REGION Network 20: UNLOCK
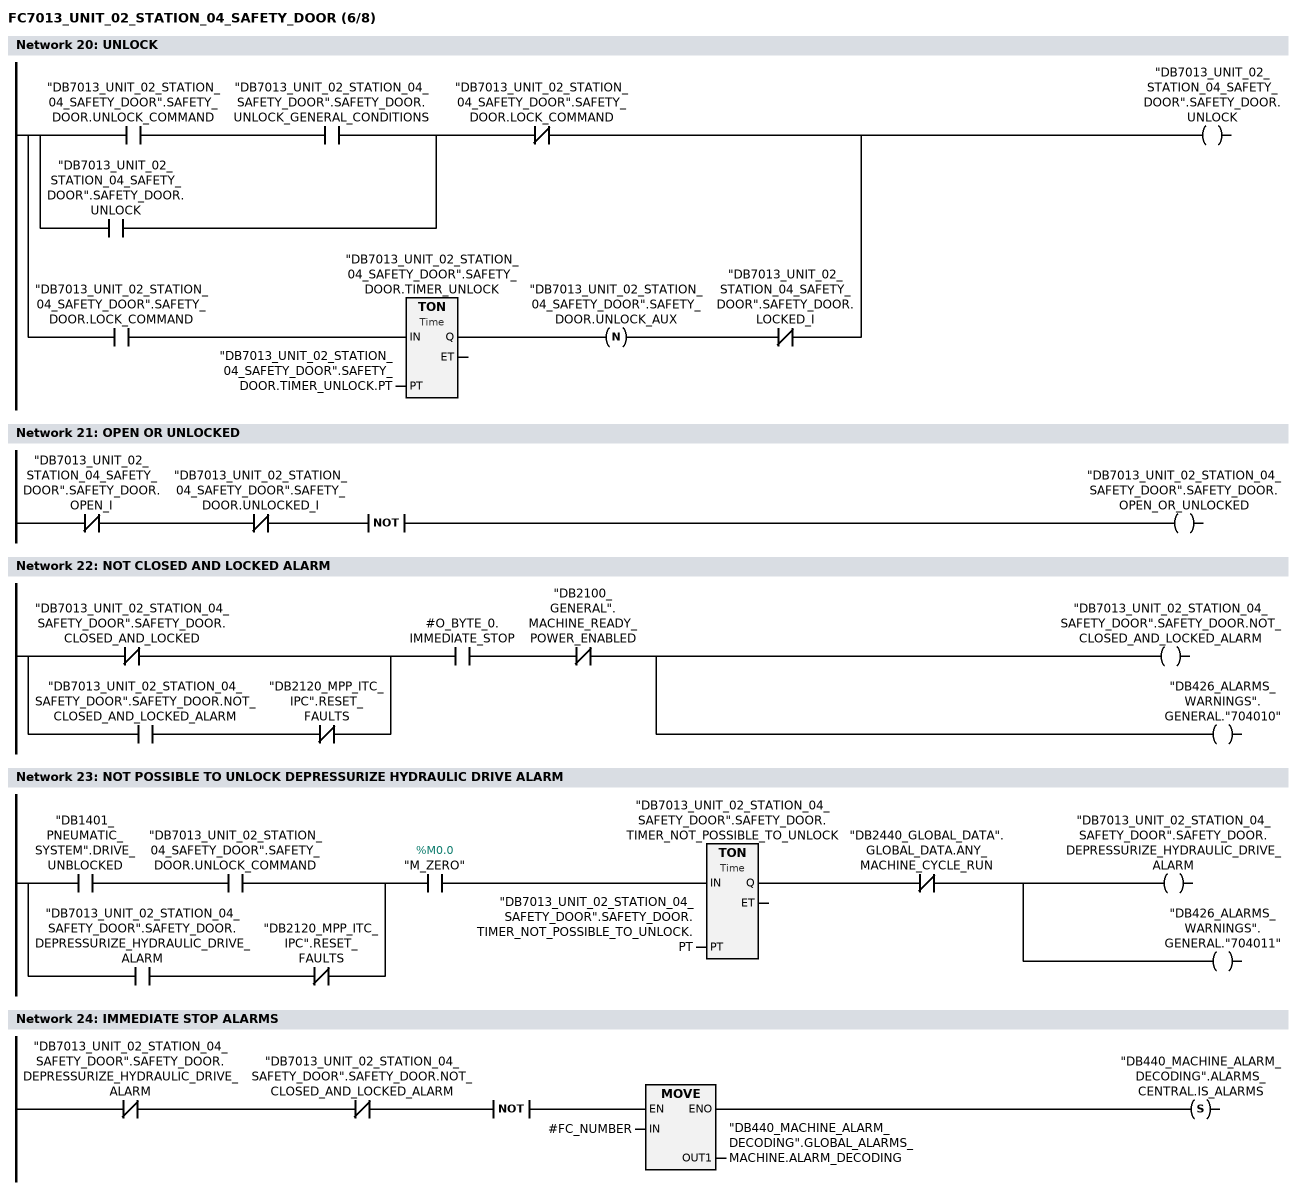
   RUNG wire#powerrail
      Contact( "DB7013_UNIT_02_STATION_04_SAFETY_DOOR".SAFETY_DOOR.UNLOCK_COMMAND )
      Contact( "DB7013_UNIT_02_STATION_04_SAFETY_DOOR".SAFETY_DOOR.UNLOCK_GENERAL_CONDITIONS )
      wire#w1
      I_Contact( "DB7013_UNIT_02_STATION_04_SAFETY_DOOR".SAFETY_DOOR.LOCK_COMMAND )
      wire#w2
      Coil( "DB7013_UNIT_02_STATION_04_SAFETY_DOOR".SAFETY_DOOR.UNLOCK )
   END_RUNG
   RUNG wire#powerrail
      Contact( "DB7013_UNIT_02_STATION_04_SAFETY_DOOR".SAFETY_DOOR.UNLOCK )
   END_RUNG wire#w1
   RUNG wire#powerrail
      Contact( "DB7013_UNIT_02_STATION_04_SAFETY_DOOR".SAFETY_DOOR.LOCK_COMMAND )
      { S7_Templates := "time_type := Time" } "DB7013_UNIT_02_STATION_04_SAFETY_DOOR".SAFETY_DOOR.TIMER_UNLOCK.TON(pt := "DB7013_UNIT_02_STATION_04_SAFETY_DOOR".SAFETY_DOOR.TIMER_UNLOCK.PT, et =>)
      N_Trig( "DB7013_UNIT_02_STATION_04_SAFETY_DOOR".SAFETY_DOOR.UNLOCK_AUX )
      I_Contact( "DB7013_UNIT_02_STATION_04_SAFETY_DOOR".SAFETY_DOOR.LOCKED_I )
   END_RUNG wire#w2
   // the same network as SCL:
   "DB7013_UNIT_02_STATION_04_SAFETY_DOOR".SAFETY_DOOR.TIMER_UNLOCK.TON(IN := "DB7013_UNIT_02_STATION_04_SAFETY_DOOR".SAFETY_DOOR.LOCK_COMMAND,
                           PT := "DB7013_UNIT_02_STATION_04_SAFETY_DOOR".SAFETY_DOOR.TIMER_UNLOCK.PT);
   #_w1 := NOT "DB7013_UNIT_02_STATION_04_SAFETY_DOOR".SAFETY_DOOR.TIMER_UNLOCK.Q AND "DB7013_UNIT_02_STATION_04_SAFETY_DOOR".SAFETY_DOOR.UNLOCK_AUX;   // falling edge
   "DB7013_UNIT_02_STATION_04_SAFETY_DOOR".SAFETY_DOOR.UNLOCK_AUX := "DB7013_UNIT_02_STATION_04_SAFETY_DOOR".SAFETY_DOOR.TIMER_UNLOCK.Q;
   "DB7013_UNIT_02_STATION_04_SAFETY_DOOR".SAFETY_DOOR.UNLOCK := ((("DB7013_UNIT_02_STATION_04_SAFETY_DOOR".SAFETY_DOOR.UNLOCK_COMMAND AND "DB7013_UNIT_02_STATION_04_SAFETY_DOOR".SAFETY_DOOR.UNLOCK_GENERAL_CONDITIONS) OR "DB7013_UNIT_02_STATION_04_SAFETY_DOOR".SAFETY_DOOR.UNLOCK) AND NOT "DB7013_UNIT_02_STATION_04_SAFETY_DOOR".SAFETY_DOOR.LOCK_COMMAND) OR (#_w1 AND NOT "DB7013_UNIT_02_STATION_04_SAFETY_DOOR".SAFETY_DOOR.LOCKED_I);
END_REGION

REGION Network 21: OPEN OR UNLOCKED
   RUNG wire#powerrail
      I_Contact( "DB7013_UNIT_02_STATION_04_SAFETY_DOOR".SAFETY_DOOR.OPEN_I )
      I_Contact( "DB7013_UNIT_02_STATION_04_SAFETY_DOOR".SAFETY_DOOR.UNLOCKED_I )
      Not()
      Coil( "DB7013_UNIT_02_STATION_04_SAFETY_DOOR".SAFETY_DOOR.OPEN_OR_UNLOCKED )
   END_RUNG
   // the same network as SCL:
   "DB7013_UNIT_02_STATION_04_SAFETY_DOOR".SAFETY_DOOR.OPEN_OR_UNLOCKED := NOT (NOT "DB7013_UNIT_02_STATION_04_SAFETY_DOOR".SAFETY_DOOR.OPEN_I AND NOT "DB7013_UNIT_02_STATION_04_SAFETY_DOOR".SAFETY_DOOR.UNLOCKED_I);
END_REGION

REGION Network 22: NOT CLOSED AND LOCKED ALARM
   RUNG wire#powerrail
      I_Contact( "DB7013_UNIT_02_STATION_04_SAFETY_DOOR".SAFETY_DOOR.CLOSED_AND_LOCKED )
      wire#w1
      Contact( #O_BYTE_0.IMMEDIATE_STOP )
      I_Contact( "DB2100_GENERAL".MACHINE_READY_POWER_ENABLED )
      wire#w2
      Coil( "DB7013_UNIT_02_STATION_04_SAFETY_DOOR".SAFETY_DOOR.NOT_CLOSED_AND_LOCKED_ALARM )
   END_RUNG
   RUNG wire#powerrail
      Contact( "DB7013_UNIT_02_STATION_04_SAFETY_DOOR".SAFETY_DOOR.NOT_CLOSED_AND_LOCKED_ALARM )
      I_Contact( "DB2120_MPP_ITC_IPC".RESET_FAULTS )
   END_RUNG wire#w1
   RUNG wire#w2
      Coil( "DB426_ALARMS_WARNINGS".GENERAL."704010" )
   END_RUNG
   // the same network as SCL:
   "DB7013_UNIT_02_STATION_04_SAFETY_DOOR".SAFETY_DOOR.NOT_CLOSED_AND_LOCKED_ALARM := (NOT "DB7013_UNIT_02_STATION_04_SAFETY_DOOR".SAFETY_DOOR.CLOSED_AND_LOCKED OR ("DB7013_UNIT_02_STATION_04_SAFETY_DOOR".SAFETY_DOOR.NOT_CLOSED_AND_LOCKED_ALARM AND NOT "DB2120_MPP_ITC_IPC".RESET_FAULTS)) AND #O_BYTE_0.IMMEDIATE_STOP AND NOT "DB2100_GENERAL".MACHINE_READY_POWER_ENABLED;
   "DB426_ALARMS_WARNINGS".GENERAL."704010" := "DB7013_UNIT_02_STATION_04_SAFETY_DOOR".SAFETY_DOOR.NOT_CLOSED_AND_LOCKED_ALARM;
END_REGION

REGION Network 23: NOT POSSIBLE TO UNLOCK DEPRESSURIZE HYDRAULIC DRIVE ALARM
   RUNG wire#powerrail
      Contact( "DB1401_PNEUMATIC_SYSTEM".DRIVE_UNBLOCKED )
      Contact( "DB7013_UNIT_02_STATION_04_SAFETY_DOOR".SAFETY_DOOR.UNLOCK_COMMAND )
      wire#w1
      Contact( "M_ZERO" )
      { S7_Templates := "time_type := Time" } "DB7013_UNIT_02_STATION_04_SAFETY_DOOR".SAFETY_DOOR.TIMER_NOT_POSSIBLE_TO_UNLOCK.TON(pt := "DB7013_UNIT_02_STATION_04_SAFETY_DOOR".SAFETY_DOOR.TIMER_NOT_POSSIBLE_TO_UNLOCK.PT, et =>)
      I_Contact( "DB2440_GLOBAL_DATA".GLOBAL_DATA.ANY_MACHINE_CYCLE_RUN )
      wire#w2
      Coil( "DB7013_UNIT_02_STATION_04_SAFETY_DOOR".SAFETY_DOOR.DEPRESSURIZE_HYDRAULIC_DRIVE_ALARM )
   END_RUNG
   RUNG wire#powerrail
      Contact( "DB7013_UNIT_02_STATION_04_SAFETY_DOOR".SAFETY_DOOR.DEPRESSURIZE_HYDRAULIC_DRIVE_ALARM )
      I_Contact( "DB2120_MPP_ITC_IPC".RESET_FAULTS )
   END_RUNG wire#w1
   RUNG wire#w2
      Coil( "DB426_ALARMS_WARNINGS".GENERAL."704011" )
   END_RUNG
   // the same network as SCL:
   "DB7013_UNIT_02_STATION_04_SAFETY_DOOR".SAFETY_DOOR.TIMER_NOT_POSSIBLE_TO_UNLOCK.TON(IN := (("DB1401_PNEUMATIC_SYSTEM".DRIVE_UNBLOCKED AND "DB7013_UNIT_02_STATION_04_SAFETY_DOOR".SAFETY_DOOR.UNLOCK_COMMAND) OR ("DB7013_UNIT_02_STATION_04_SAFETY_DOOR".SAFETY_DOOR.DEPRESSURIZE_HYDRAULIC_DRIVE_ALARM AND NOT "DB2120_MPP_ITC_IPC".RESET_FAULTS)) AND "M_ZERO",
                           PT := "DB7013_UNIT_02_STATION_04_SAFETY_DOOR".SAFETY_DOOR.TIMER_NOT_POSSIBLE_TO_UNLOCK.PT);
   "DB7013_UNIT_02_STATION_04_SAFETY_DOOR".SAFETY_DOOR.DEPRESSURIZE_HYDRAULIC_DRIVE_ALARM := "DB7013_UNIT_02_STATION_04_SAFETY_DOOR".SAFETY_DOOR.TIMER_NOT_POSSIBLE_TO_UNLOCK.Q AND NOT "DB2440_GLOBAL_DATA".GLOBAL_DATA.ANY_MACHINE_CYCLE_RUN;
   "DB426_ALARMS_WARNINGS".GENERAL."704011" := "DB7013_UNIT_02_STATION_04_SAFETY_DOOR".SAFETY_DOOR.DEPRESSURIZE_HYDRAULIC_DRIVE_ALARM;
END_REGION

REGION Network 24: IMMEDIATE STOP ALARMS
   RUNG wire#powerrail
      I_Contact( "DB7013_UNIT_02_STATION_04_SAFETY_DOOR".SAFETY_DOOR.DEPRESSURIZE_HYDRAULIC_DRIVE_ALARM )
      I_Contact( "DB7013_UNIT_02_STATION_04_SAFETY_DOOR".SAFETY_DOOR.NOT_CLOSED_AND_LOCKED_ALARM )
      Not()
      { S7_GenerateENO := "TRUE" } Move(in := #FC_NUMBER, out1 => "DB440_MACHINE_ALARM_DECODING".GLOBAL_ALARMS_MACHINE.ALARM_DECODING)
      S_Coil( "DB440_MACHINE_ALARM_DECODING".ALARMS_CENTRAL.IS_ALARMS )
   END_RUNG
   // the same network as SCL:
   // ENO of a box is taken as its EN; it also drops when the box reports an error
   IF NOT (NOT "DB7013_UNIT_02_STATION_04_SAFETY_DOOR".SAFETY_DOOR.DEPRESSURIZE_HYDRAULIC_DRIVE_ALARM AND NOT "DB7013_UNIT_02_STATION_04_SAFETY_DOOR".SAFETY_DOOR.NOT_CLOSED_AND_LOCKED_ALARM) THEN
       "DB440_MACHINE_ALARM_DECODING".GLOBAL_ALARMS_MACHINE.ALARM_DECODING := #FC_NUMBER;
       "DB440_MACHINE_ALARM_DECODING".ALARMS_CENTRAL.IS_ALARMS := TRUE;
   END_IF;
END_REGION

REGION Network 25: UNLOCK REQUEST WARNING
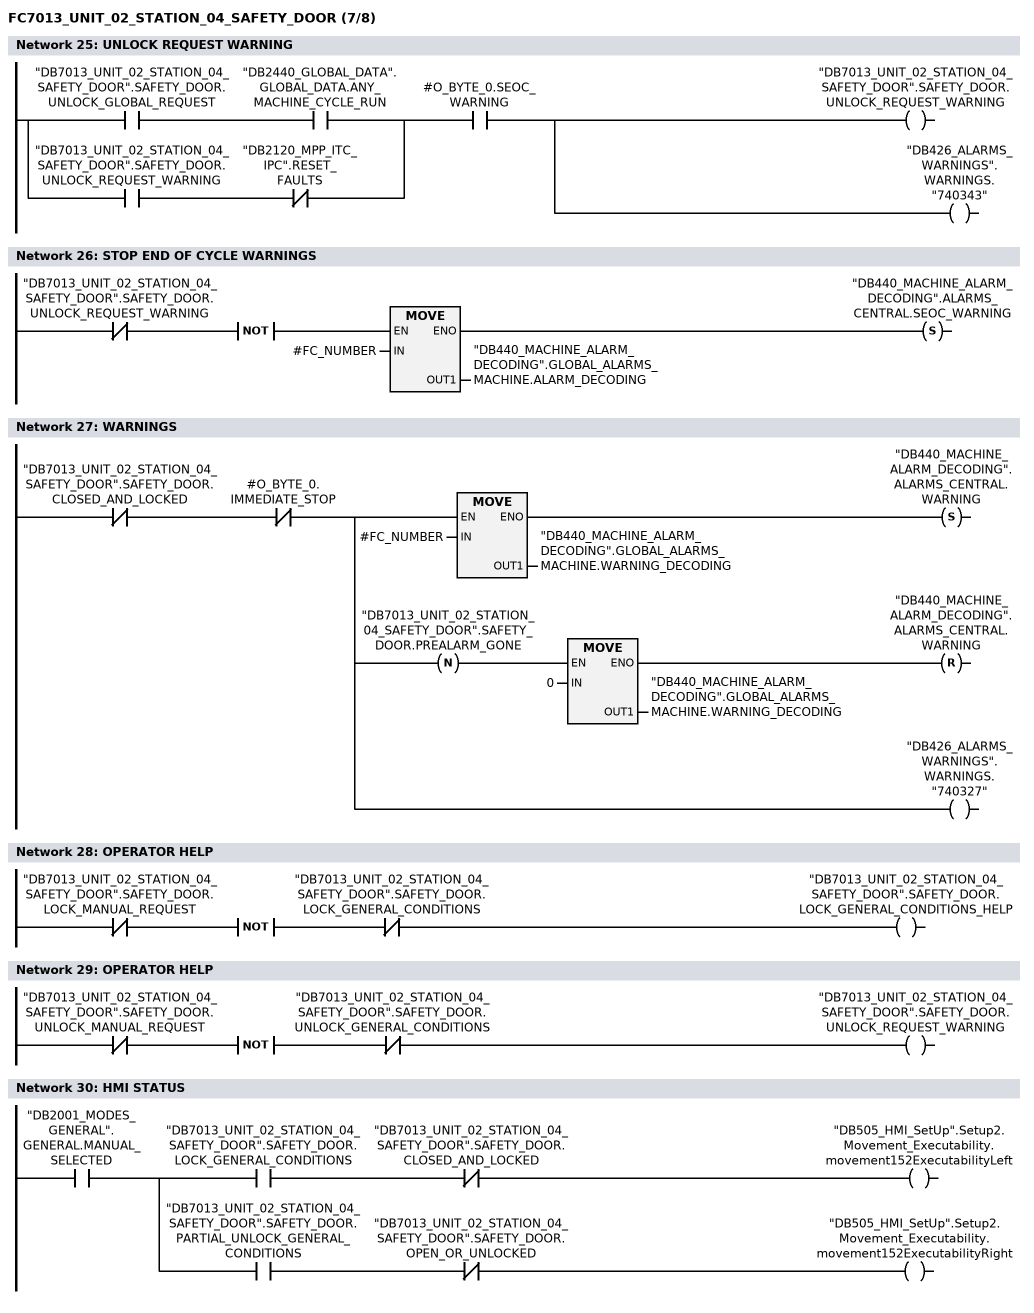
   RUNG wire#powerrail
      Contact( "DB7013_UNIT_02_STATION_04_SAFETY_DOOR".SAFETY_DOOR.UNLOCK_GLOBAL_REQUEST )
      Contact( "DB2440_GLOBAL_DATA".GLOBAL_DATA.ANY_MACHINE_CYCLE_RUN )
      wire#w1
      Contact( #O_BYTE_0.SEOC_WARNING )
      wire#w2
      Coil( "DB7013_UNIT_02_STATION_04_SAFETY_DOOR".SAFETY_DOOR.UNLOCK_REQUEST_WARNING )
   END_RUNG
   RUNG wire#powerrail
      Contact( "DB7013_UNIT_02_STATION_04_SAFETY_DOOR".SAFETY_DOOR.UNLOCK_REQUEST_WARNING )
      I_Contact( "DB2120_MPP_ITC_IPC".RESET_FAULTS )
   END_RUNG wire#w1
   RUNG wire#w2
      Coil( "DB426_ALARMS_WARNINGS".WARNINGS."740343" )
   END_RUNG
   // the same network as SCL:
   "DB7013_UNIT_02_STATION_04_SAFETY_DOOR".SAFETY_DOOR.UNLOCK_REQUEST_WARNING := (("DB7013_UNIT_02_STATION_04_SAFETY_DOOR".SAFETY_DOOR.UNLOCK_GLOBAL_REQUEST AND "DB2440_GLOBAL_DATA".GLOBAL_DATA.ANY_MACHINE_CYCLE_RUN) OR ("DB7013_UNIT_02_STATION_04_SAFETY_DOOR".SAFETY_DOOR.UNLOCK_REQUEST_WARNING AND NOT "DB2120_MPP_ITC_IPC".RESET_FAULTS)) AND #O_BYTE_0.SEOC_WARNING;
   "DB426_ALARMS_WARNINGS".WARNINGS."740343" := "DB7013_UNIT_02_STATION_04_SAFETY_DOOR".SAFETY_DOOR.UNLOCK_REQUEST_WARNING;
END_REGION

REGION Network 26: STOP END OF CYCLE WARNINGS
   RUNG wire#powerrail
      I_Contact( "DB7013_UNIT_02_STATION_04_SAFETY_DOOR".SAFETY_DOOR.UNLOCK_REQUEST_WARNING )
      Not()
      { S7_GenerateENO := "TRUE" } Move(in := #FC_NUMBER, out1 => "DB440_MACHINE_ALARM_DECODING".GLOBAL_ALARMS_MACHINE.ALARM_DECODING)
      S_Coil( "DB440_MACHINE_ALARM_DECODING".ALARMS_CENTRAL.SEOC_WARNING )
   END_RUNG
   // the same network as SCL:
   // ENO of a box is taken as its EN; it also drops when the box reports an error
   IF NOT (NOT "DB7013_UNIT_02_STATION_04_SAFETY_DOOR".SAFETY_DOOR.UNLOCK_REQUEST_WARNING) THEN
       "DB440_MACHINE_ALARM_DECODING".GLOBAL_ALARMS_MACHINE.ALARM_DECODING := #FC_NUMBER;
       "DB440_MACHINE_ALARM_DECODING".ALARMS_CENTRAL.SEOC_WARNING := TRUE;
   END_IF;
END_REGION

REGION Network 27: WARNINGS
   RUNG wire#powerrail
      I_Contact( "DB7013_UNIT_02_STATION_04_SAFETY_DOOR".SAFETY_DOOR.CLOSED_AND_LOCKED )
      I_Contact( #O_BYTE_0.IMMEDIATE_STOP )
      wire#w1
      { S7_GenerateENO := "TRUE" } Move(in := #FC_NUMBER, out1 => "DB440_MACHINE_ALARM_DECODING".GLOBAL_ALARMS_MACHINE.WARNING_DECODING)
      S_Coil( "DB440_MACHINE_ALARM_DECODING".ALARMS_CENTRAL.WARNING )
   END_RUNG
   RUNG wire#w1
      N_Trig( "DB7013_UNIT_02_STATION_04_SAFETY_DOOR".SAFETY_DOOR.PREALARM_GONE )
      { S7_GenerateENO := "TRUE" } Move(in := 0, out1 => "DB440_MACHINE_ALARM_DECODING".GLOBAL_ALARMS_MACHINE.WARNING_DECODING)
      R_Coil( "DB440_MACHINE_ALARM_DECODING".ALARMS_CENTRAL.WARNING )
   END_RUNG
   RUNG wire#w1
      Coil( "DB426_ALARMS_WARNINGS".WARNINGS."740327" )
   END_RUNG
   // the same network as SCL:
   // ENO of a box is taken as its EN; it also drops when the box reports an error
   #_w1 := NOT "DB7013_UNIT_02_STATION_04_SAFETY_DOOR".SAFETY_DOOR.CLOSED_AND_LOCKED AND NOT #O_BYTE_0.IMMEDIATE_STOP;
   IF #_w1 THEN
       "DB440_MACHINE_ALARM_DECODING".GLOBAL_ALARMS_MACHINE.WARNING_DECODING := #FC_NUMBER;
       "DB440_MACHINE_ALARM_DECODING".ALARMS_CENTRAL.WARNING := TRUE;
   END_IF;
   #_w2 := NOT #_w1 AND "DB7013_UNIT_02_STATION_04_SAFETY_DOOR".SAFETY_DOOR.PREALARM_GONE;   // falling edge
   "DB7013_UNIT_02_STATION_04_SAFETY_DOOR".SAFETY_DOOR.PREALARM_GONE := #_w1;
   IF #_w2 THEN
       "DB440_MACHINE_ALARM_DECODING".GLOBAL_ALARMS_MACHINE.WARNING_DECODING := 0;
       "DB440_MACHINE_ALARM_DECODING".ALARMS_CENTRAL.WARNING := FALSE;
   END_IF;
   "DB426_ALARMS_WARNINGS".WARNINGS."740327" := #_w1;
END_REGION

REGION Network 28: OPERATOR HELP
   RUNG wire#powerrail
      I_Contact( "DB7013_UNIT_02_STATION_04_SAFETY_DOOR".SAFETY_DOOR.LOCK_MANUAL_REQUEST )
      Not()
      I_Contact( "DB7013_UNIT_02_STATION_04_SAFETY_DOOR".SAFETY_DOOR.LOCK_GENERAL_CONDITIONS )
      Coil( "DB7013_UNIT_02_STATION_04_SAFETY_DOOR".SAFETY_DOOR.LOCK_GENERAL_CONDITIONS_HELP )
   END_RUNG
   // the same network as SCL:
   "DB7013_UNIT_02_STATION_04_SAFETY_DOOR".SAFETY_DOOR.LOCK_GENERAL_CONDITIONS_HELP := NOT (NOT "DB7013_UNIT_02_STATION_04_SAFETY_DOOR".SAFETY_DOOR.LOCK_MANUAL_REQUEST) AND NOT "DB7013_UNIT_02_STATION_04_SAFETY_DOOR".SAFETY_DOOR.LOCK_GENERAL_CONDITIONS;
END_REGION

REGION Network 29: OPERATOR HELP
   RUNG wire#powerrail
      I_Contact( "DB7013_UNIT_02_STATION_04_SAFETY_DOOR".SAFETY_DOOR.UNLOCK_MANUAL_REQUEST )
      Not()
      I_Contact( "DB7013_UNIT_02_STATION_04_SAFETY_DOOR".SAFETY_DOOR.UNLOCK_GENERAL_CONDITIONS )
      Coil( "DB7013_UNIT_02_STATION_04_SAFETY_DOOR".SAFETY_DOOR.UNLOCK_REQUEST_WARNING )
   END_RUNG
   // the same network as SCL:
   "DB7013_UNIT_02_STATION_04_SAFETY_DOOR".SAFETY_DOOR.UNLOCK_REQUEST_WARNING := NOT (NOT "DB7013_UNIT_02_STATION_04_SAFETY_DOOR".SAFETY_DOOR.UNLOCK_MANUAL_REQUEST) AND NOT "DB7013_UNIT_02_STATION_04_SAFETY_DOOR".SAFETY_DOOR.UNLOCK_GENERAL_CONDITIONS;
END_REGION

REGION Network 30: HMI STATUS
   RUNG wire#powerrail
      Contact( "DB2001_MODES_GENERAL".GENERAL.MANUAL_SELECTED )
      wire#w1
      Contact( "DB7013_UNIT_02_STATION_04_SAFETY_DOOR".SAFETY_DOOR.LOCK_GENERAL_CONDITIONS )
      I_Contact( "DB7013_UNIT_02_STATION_04_SAFETY_DOOR".SAFETY_DOOR.CLOSED_AND_LOCKED )
      Coil( "DB505_HMI_SetUp".Setup2.Movement_Executability.movement152ExecutabilityLeft )
   END_RUNG
   RUNG wire#w1
      Contact( "DB7013_UNIT_02_STATION_04_SAFETY_DOOR".SAFETY_DOOR.PARTIAL_UNLOCK_GENERAL_CONDITIONS )
      I_Contact( "DB7013_UNIT_02_STATION_04_SAFETY_DOOR".SAFETY_DOOR.OPEN_OR_UNLOCKED )
      Coil( "DB505_HMI_SetUp".Setup2.Movement_Executability.movement152ExecutabilityRight )
   END_RUNG
   // the same network as SCL:
   "DB505_HMI_SetUp".Setup2.Movement_Executability.movement152ExecutabilityLeft := "DB2001_MODES_GENERAL".GENERAL.MANUAL_SELECTED AND "DB7013_UNIT_02_STATION_04_SAFETY_DOOR".SAFETY_DOOR.LOCK_GENERAL_CONDITIONS AND NOT "DB7013_UNIT_02_STATION_04_SAFETY_DOOR".SAFETY_DOOR.CLOSED_AND_LOCKED;
   "DB505_HMI_SetUp".Setup2.Movement_Executability.movement152ExecutabilityRight := "DB2001_MODES_GENERAL".GENERAL.MANUAL_SELECTED AND "DB7013_UNIT_02_STATION_04_SAFETY_DOOR".SAFETY_DOOR.PARTIAL_UNLOCK_GENERAL_CONDITIONS AND NOT "DB7013_UNIT_02_STATION_04_SAFETY_DOOR".SAFETY_DOOR.OPEN_OR_UNLOCKED;
END_REGION

REGION Network 31: HMI STATUS
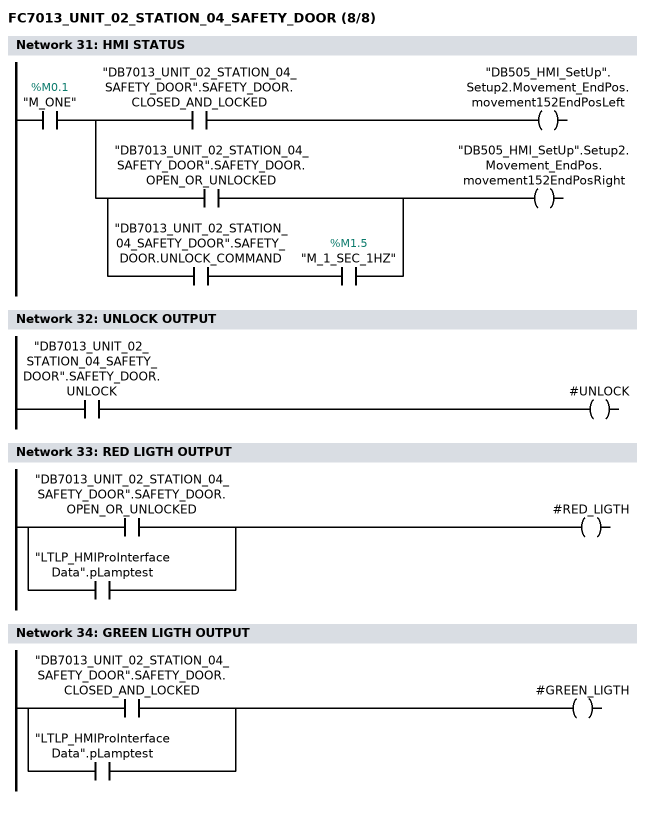
   RUNG wire#powerrail
      Contact( "M_ONE" )
      wire#w1
      Contact( "DB7013_UNIT_02_STATION_04_SAFETY_DOOR".SAFETY_DOOR.CLOSED_AND_LOCKED )
      Coil( "DB505_HMI_SetUp".Setup2.Movement_EndPos.movement152EndPosLeft )
   END_RUNG
   RUNG wire#w1
      Contact( "DB7013_UNIT_02_STATION_04_SAFETY_DOOR".SAFETY_DOOR.OPEN_OR_UNLOCKED )
      wire#w2
      Coil( "DB505_HMI_SetUp".Setup2.Movement_EndPos.movement152EndPosRight )
   END_RUNG
   RUNG wire#w1
      Contact( "DB7013_UNIT_02_STATION_04_SAFETY_DOOR".SAFETY_DOOR.UNLOCK_COMMAND )
      Contact( "M_1_SEC_1HZ" )
   END_RUNG wire#w2
   // the same network as SCL:
   "DB505_HMI_SetUp".Setup2.Movement_EndPos.movement152EndPosLeft := "M_ONE" AND "DB7013_UNIT_02_STATION_04_SAFETY_DOOR".SAFETY_DOOR.CLOSED_AND_LOCKED;
   "DB505_HMI_SetUp".Setup2.Movement_EndPos.movement152EndPosRight := "M_ONE" AND ("DB7013_UNIT_02_STATION_04_SAFETY_DOOR".SAFETY_DOOR.OPEN_OR_UNLOCKED OR ("DB7013_UNIT_02_STATION_04_SAFETY_DOOR".SAFETY_DOOR.UNLOCK_COMMAND AND "M_1_SEC_1HZ"));
END_REGION

REGION Network 32: UNLOCK OUTPUT
   RUNG wire#powerrail
      Contact( "DB7013_UNIT_02_STATION_04_SAFETY_DOOR".SAFETY_DOOR.UNLOCK )
      Coil( #UNLOCK )
   END_RUNG
   // the same network as SCL:
   #UNLOCK := "DB7013_UNIT_02_STATION_04_SAFETY_DOOR".SAFETY_DOOR.UNLOCK;
END_REGION

REGION Network 33: RED LIGTH OUTPUT
   RUNG wire#powerrail
      Contact( "DB7013_UNIT_02_STATION_04_SAFETY_DOOR".SAFETY_DOOR.OPEN_OR_UNLOCKED )
      wire#w1
      Coil( #RED_LIGTH )
   END_RUNG
   RUNG wire#powerrail
      Contact( "LTLP_HMIProInterfaceData".pLamptest )
   END_RUNG wire#w1
   // the same network as SCL:
   #RED_LIGTH := "DB7013_UNIT_02_STATION_04_SAFETY_DOOR".SAFETY_DOOR.OPEN_OR_UNLOCKED OR "LTLP_HMIProInterfaceData".pLamptest;
END_REGION

REGION Network 34: GREEN LIGTH OUTPUT
   RUNG wire#powerrail
      Contact( "DB7013_UNIT_02_STATION_04_SAFETY_DOOR".SAFETY_DOOR.CLOSED_AND_LOCKED )
      wire#w1
      Coil( #GREEN_LIGTH )
   END_RUNG
   RUNG wire#powerrail
      Contact( "LTLP_HMIProInterfaceData".pLamptest )
   END_RUNG wire#w1
   // the same network as SCL:
   #GREEN_LIGTH := "DB7013_UNIT_02_STATION_04_SAFETY_DOOR".SAFETY_DOOR.CLOSED_AND_LOCKED OR "LTLP_HMIProInterfaceData".pLamptest;
END_REGION
END_FUNCTION

FUNCTION "FC8007_UNIT_03_PART_STATUS_FULL_DEPTH" : Void   // FC8007, LAD
{ S7_Optimized_Access := 'TRUE' }
VERSION : 0.1
// stored: AutoNumber false, IsIECCheckEnabled false, SetENOAutomatically false, UDAEnableTagReadback false
BEGIN

REGION Network 1: FIXTURE 1 PART STATUS UNIT 01
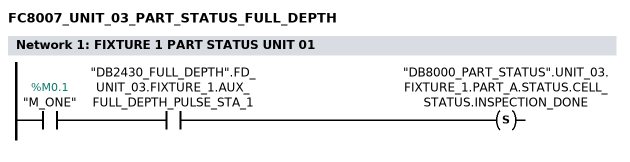
   RUNG wire#powerrail
      Contact( "M_ONE" )
      Contact( "DB2430_FULL_DEPTH".FD_UNIT_03.FIXTURE_1.AUX_FULL_DEPTH_PULSE_STA_1 )
      S_Coil( "DB8000_PART_STATUS".UNIT_03.FIXTURE_1.PART_A.STATUS.CELL_STATUS.INSPECTION_DONE )
   END_RUNG
   // the same network as SCL:
   IF "M_ONE" AND "DB2430_FULL_DEPTH".FD_UNIT_03.FIXTURE_1.AUX_FULL_DEPTH_PULSE_STA_1 THEN
       "DB8000_PART_STATUS".UNIT_03.FIXTURE_1.PART_A.STATUS.CELL_STATUS.INSPECTION_DONE := TRUE;
   END_IF;
END_REGION
END_FUNCTION

FUNCTION_BLOCK "FB2105_PSE200U_SITOP"
{ S7_Optimized_Access := 'FALSE' }
AUTHOR : DFCS
FAMILY : SITOP
NAME : PSE200U
VERSION : 2.3
   VAR_INPUT 
      impulse : Bool;
      reset : Bool;
   END_VAR

   VAR_OUTPUT 
      done : Bool;
      busy : Bool;
      channelState : Byte;
      status : Word;
      error : Bool;
   END_VAR

   VAR 
      statImpulseOld : Bool;
      statResetOld : Bool;
      statTimeSaver : Struct
         TimeTckRisingEdge : Time;
         TimeTckFallingEdge : Time;
         RisingEdgeDetected : Bool;
         FallingEdgeDetected : Bool;
         stateEdge : Int;
      END_STRUCT;
      statDeltaTimeImpulse : Time;
      statDeltaTimePause : Time;
      statStartImpulseDetected : Bool;
      statImpulseDetected : Bool;
      statChannelState : Byte;
      statChannelStateBool { ExternalAccessible := 'False'; ExternalVisible := 'False'; ExternalWritable := 'False'} AT statChannelState : Array[0..7] of Bool;
      statTimePauseSave0 : Time;
      statTimePauseSave1 : Time;
      statTimePauseSave2 : Time;
      statTimePauseSave3 : Time;
      statTimePauseSave4 : Time;
      statTimeImpulseSave0 : Time;
      statTimeImpulseSave1 : Time;
      statTimeImpulseSave2 : Time;
      statTimeImpulseSave3 : Time;
      statTimeImpulseSave4 : Time;
      statFrameImulseDetected : Bool;
      statNumberOfImpulses : Int;
      statChannelActive1 : Bool;
      statChannelActive2 : Bool;
      statChannelActive3 : Bool;
      statChannelActive4 : Bool;
      statCountChannelPos : Int;
      statCurrentPos1 : Int;
      statCurrentPos2 : Int;
      statCurrentPos3 : Int;
      statCurrentPos4 : Int;
      statTimeToImpulse : Time;
      statTimePause : Time;
      statTimeImpulse : Time;
      statTimeFrame : Time;
      statFrameOk : Bool;
      statCycleTimeNok : Bool;
      statSysTime : Time;
      statSysTimeOld : Time;
      statDeltaSysTime : Time;
      instSysTimer {InstructionName := 'TON_TIME'; LibVersion := '1.0'} : TON_TIME;
      statSysTimerStart : Bool;
      statStatus : Word;
      statIndex : Int;
      statSysTimerRun : Time;
      instWatchDogTimerR {InstructionName := 'TON_TIME'; LibVersion := '1.0'} : TON_TIME;
      statWatchDogTimerStartR : Bool;
      statWatchDogTimerRunR : Time;
      instWatchDogTimerF {InstructionName := 'TON_TIME'; LibVersion := '1.0'} : TON_TIME;
      statWatchDogTimerStartF : Bool;
      statWatchDogTimerRunF : Time;
      statResetRequest : Bool;
   END_VAR

   VAR_TEMP 
      tempLatchTime : Time;
   END_VAR

   VAR CONSTANT 
      STATE_IDLE : Int := 0;
      STATE_EVALUATION : Int := 1;
      STATE_ERROR : Int := 2;
      TIME_FRAME_MAX : Time := T#2S_850MS;
      TIME_FRAME_MIN : Time := T#2S_650MS;
      TIME_STARTIMPULSE_MIN : Time := T#400MS;
      TIME_STARTIMPULSE_MAX : Time := T#600MS;
      TIME_IMPULSE_MIN : Time := T#150MS;
      TIME_IMPULSE_MAX : Time := T#350MS;
      TIME_PAUSE1_MIN : Time := T#150MS;
      TIME_PAUSE1_MAX : Time := T#350MS;
      TIME_PAUSE2_MIN : Time := T#650MS;
      TIME_PAUSE2_MAX : Time := T#850MS;
      TIME_PAUSE3_MIN : Time := T#1S_150MS;
      TIME_PAUSE3_MAX : Time := T#1S_350MS;
      TIME_PAUSE4_MIN : Time := T#1S_650MS;
      TIME_PAUSE4_MAX : Time := T#1S_850MS;
      TIME_PAUSE_FRAME_MIN : Time := T#2S_150MS;
      TIME_PAUSE_FRAME_MAX : Time := T#2S_350MS;
   END_VAR


BEGIN
	   
	    // Calculate cycle time
	    #statSysTime := TIME_TCK();
	    #statDeltaSysTime := #statSysTime - #statSysTimeOld;
	    
	    IF (#statDeltaSysTime < t#0ms)
	    THEN
	        #statDeltaSysTime := #statDeltaSysTime + T#2147483647ms;
	        
	        IF #statDeltaSysTime < t#0ms
	        THEN
	            #statCycleTimeNok := true;
	            #statSysTimeOld := #statSysTime;
	            RETURN;
	        ELSE
	            #statCycleTimeNok := false;
	        END_IF;
	        
	    ELSIF #statDeltaSysTime >= t#102ms
	    THEN
	        #statCycleTimeNok := true;
	        #statSysTimerStart := true;
	    ELSE
	        #statCycleTimeNok := false;
	        #statSysTimerStart := false;
	    END_IF;
	    
	    //REGION edgeDetection
	        
	        IF ((#reset = true)
	            AND (#statResetOld = false))
	        THEN
	            #statSysTimerStart := false;
	            #statWatchDogTimerStartR := false;
	            #statWatchDogTimerStartF := false;
	            #statResetRequest := true;
	            #statIndex := #STATE_IDLE;
	        END_IF;
	        
	        //Rising edge at impulse input
	        IF ((#impulse = True)
	            AND (#statImpulseOld = False))
	        THEN
	            #tempLatchTime := TIME_TCK();
	            #statTimeSaver.RisingEdgeDetected := true;
	            #statTimeSaver.stateEdge := 15;
	            #statTimeSaver.TimeTckRisingEdge := #tempLatchTime;
	            #statWatchDogTimerStartR := true;
	            #statWatchDogTimerStartF := false;
	            
	            IF (#busy = false) THEN
	        
	                #busy := true;
	                #done := false;
	                #error := false;
	                #status := 16#0000;
	            END_IF;
	
	            
	            IF #statCycleTimeNok = false
	                AND #statResetRequest = false
	            THEN
	                #statIndex := #STATE_EVALUATION;
	            END_IF;
	        END_IF;
	        
	        //Falling edge at impulse input
	        IF ((#impulse = False)
	            AND (#statImpulseOld = True))
	        THEN
	            #tempLatchTime := TIME_TCK();
	            #statTimeSaver.FallingEdgeDetected := true;
	            #statTimeSaver.stateEdge := 16;
	            #statTimeSaver.TimeTckFallingEdge := #tempLatchTime;
	            #statWatchDogTimerStartF:=true;
	            #statWatchDogTimerStartR:=false;
	            
	            IF #statCycleTimeNok = FALSE
	                AND #statResetRequest = false
	            THEN
	                #statIndex := #STATE_EVALUATION;
	            END_IF;
	        END_IF;
	        
	        
	    //END_REGION
	    
	    IF #statTimeSaver.FallingEdgeDetected = false AND
	        #statTimeSaver.RisingEdgeDetected = FALSE
	    THEN
	        #statWatchDogTimerStartR := true;
	        #statWatchDogTimerStartF := true;
	    END_IF;
	    
	    CASE #statIndex OF
	        #STATE_IDLE:  // IDLE_STATE
	            #done := false;
	            #error := false;
	            #busy := false;
	            #status := 16#0000;
	            #statStatus := 16#0000;
	            #channelState := 16#00;
	            #statChannelState := 16#00;
	            #statFrameOk := false;
	            #statCycleTimeNok := false;
	            #statStartImpulseDetected := false;
	            #statFrameImulseDetected := false;
	            #statResetRequest := false;
	            #statTimeSaver.RisingEdgeDetected:=false;
	            #statTimeSaver.FallingEdgeDetected:=false;
	            
	        #STATE_EVALUATION:  //State: impulse detection
	            
	            //Delta time calculation
	            IF ((#statTimeSaver.RisingEdgeDetected = True)
	                AND (#statTimeSaver.FallingEdgeDetected = True))
	            THEN
	                
	                IF #statTimeSaver.stateEdge = 15 //pos. edge, evaluate delta pause
	                THEN
	                    #statDeltaTimePause := #statTimeSaver.TimeTckRisingEdge - #statTimeSaver.TimeTckFallingEdge;
	                    
	                    IF (#statDeltaTimePause < t#0ms)
	                    THEN
	                        #statDeltaTimePause := #statDeltaTimePause + T#2147483647ms;
	                        
	                        IF (#statDeltaTimePause < t#0ms)
	                        THEN
	                            #statIndex := #STATE_IDLE;
	                            #statTimeSaver.FallingEdgeDetected := false;
	                            RETURN;
	                        END_IF;
	                        
	                    ELSIF (#statDeltaTimePause > #TIME_FRAME_MAX)
	                    THEN
	                        #statIndex := #STATE_IDLE;
	                        #statTimeSaver.FallingEdgeDetected := false;
	                        RETURN;
	                    END_IF;
	                    #statTimeSaver.FallingEdgeDetected := false;
	                END_IF;
	                
	                IF #statTimeSaver.stateEdge = 16 // neg. edge, evaluate delta impulse
	                THEN
	                    #statImpulseDetected := true;
	                    #statDeltaTimeImpulse := #statTimeSaver.TimeTckFallingEdge - #statTimeSaver.TimeTckRisingEdge;
	                    
	                    IF (#statDeltaTimeImpulse < t#0ms)
	                    THEN
	                        #statDeltaTimeImpulse := #statDeltaTimeImpulse + T#2147483647ms;
	                        
	                        IF (#statDeltaTimeImpulse < t#0ms)
	                        THEN
	                            #statIndex := #STATE_IDLE;
	                            #statTimeSaver.RisingEdgeDetected := false;
	                            RETURN;
	                        END_IF;
	                        
	                    ELSIF (#statDeltaTimeImpulse > #TIME_FRAME_MAX)
	                    THEN
	                        #statIndex := #STATE_IDLE;
	                        #statTimeSaver.RisingEdgeDetected := false;
	                        RETURN;
	                    END_IF;
	                    #statTimeSaver.RisingEdgeDetected := false;
	                END_IF;
	            END_IF;
	            
	            //Start bit detection
	            IF ((#statDeltaTimeImpulse >= #TIME_STARTIMPULSE_MIN)
	                AND (#statDeltaTimeImpulse <= #TIME_STARTIMPULSE_MAX))
	                AND (#statImpulseDetected = True)
	            THEN
	                #statImpulseDetected := False;
	                #statNumberOfImpulses := 0;
	                #statCountChannelPos := 0;
	                
	                IF #statCurrentPos1 = 0
	                THEN
	                    #statTimeImpulseSave1 := t#0ms;
	                    #statTimePauseSave1 := t#0ms;
	                END_IF;
	                
	                IF #statCurrentPos2 = 0
	                THEN
	                    #statTimeImpulseSave2 := t#0ms;
	                    #statTimePauseSave2 := t#0ms;
	                END_IF;
	                
	                IF #statCurrentPos3 = 0
	                THEN
	                    #statTimeImpulseSave3 := t#0ms;
	                    #statTimePauseSave3 := t#0ms;
	                END_IF;
	                
	                IF #statCurrentPos4 = 0
	                THEN
	                    #statTimeImpulseSave4 := t#0ms;
	                    #statTimePauseSave4 := t#0ms;
	                END_IF;
	                
	                #statTimePauseSave0 := #statDeltaTimePause;
	                #statTimeImpulseSave0 := #statDeltaTimeImpulse;
	                
	                // get time in sum of imulses
	                #statTimeImpulse := #statTimeImpulseSave0 + #statTimeImpulseSave1 + #statTimeImpulseSave2 + #statTimeImpulseSave3 + #statTimeImpulseSave4;
	                
	                //get time in sum of pauses
	                #statTimePause := #statTimePauseSave0 + #statTimePauseSave1 + #statTimePauseSave2 + #statTimePauseSave3 + #statTimePauseSave4;
	                
	                // get length of frame
	                #statTimeFrame := #statTimeImpulse + #statTimePause;
	                
	                IF (#statTimeFrame >= t#2650ms)
	                    AND (#statTimeFrame <= #TIME_FRAME_MAX)
	                    AND (#statTimeToImpulse <= #TIME_FRAME_MIN)
	                THEN
	                    #statFrameOk := true;
	                END_IF;
	                
	                IF #statFrameOk = TRUE
	                    AND #statCycleTimeNok = FALSE
	                THEN
	                    // Daten Ã¼bernehmen
	                    #done := true;
	                    #busy := false;
	                    #statFrameOk := false;
	                    
	                    IF #statChannelActive1 = true
	                    THEN
	                        #statChannelStateBool[0] := false;
	                    ELSE
	                        #statChannelStateBool[0] := true;
	                    END_IF;
	                    
	                    IF #statChannelActive2 = true
	                    THEN
	                        #statChannelStateBool[1] := false;
	                    ELSE
	                        #statChannelStateBool[1] := true;
	                    END_IF;
	                    
	                    IF #statChannelActive3 = true
	                    THEN
	                        #statChannelStateBool[2] := false;
	                    ELSE
	                        #statChannelStateBool[2] := true;
	                    END_IF;
	                    
	                    IF #statChannelActive4 = true
	                    THEN
	                        #statChannelStateBool[3] := false;
	                    ELSE
	                        #statChannelStateBool[3] := true;
	                    END_IF;
	                    
	                    #channelState := #statChannelState;
	                END_IF;
	                
	                
	                // channel 4 ok
	                IF (#statDeltaTimePause >= #TIME_PAUSE1_MIN) AND
	                    (#statDeltaTimePause <= #TIME_PAUSE1_MAX)
	                THEN
	                    #statChannelActive4 := true;
	                    // channel 4 ok not ok
	                ELSIF
	                    (#statDeltaTimePause >= #TIME_PAUSE2_MIN) AND
	                    (#statDeltaTimePause <= #TIME_PAUSE2_MAX)
	                THEN
	                    #statChannelActive4 := false;
	                    // channel 3 and 4 not ok    
	                ELSIF
	                    (#statDeltaTimePause >= #TIME_PAUSE3_MIN) AND
	                    (#statDeltaTimePause <= #TIME_PAUSE3_MAX)
	                THEN
	                    #statChannelActive3 := false;
	                    #statChannelActive4 := false;
	                    // channel 2, 3, 4 not ok
	                ELSIF
	                    (#statDeltaTimePause >= #TIME_PAUSE4_MIN) AND
	                    (#statDeltaTimePause <= #TIME_PAUSE4_MAX)
	                THEN
	                    #statChannelActive2 := false;
	                    #statChannelActive3 := false;
	                    #statChannelActive4 := false;
	                    // channel 1, 2, 3, 4 not ok
	                ELSIF
	                    (#statDeltaTimePause >= #TIME_PAUSE_FRAME_MIN) AND
	                    (#statDeltaTimePause <= #TIME_PAUSE_FRAME_MAX)
	                THEN
	                    #statChannelActive1 := false;
	                    #statChannelActive2 := false;
	                    #statChannelActive3 := false;
	                    #statChannelActive4 := false;
	                END_IF;
	                
	                #statCountChannelPos := 4;
	                
	                #statCurrentPos1 := 0;
	                #statCurrentPos2 := 0;
	                #statCurrentPos3 := 0;
	                #statCurrentPos4 := 0;
	                
	                // Imulse bit detection
	            ELSIF ((#statDeltaTimeImpulse >= #TIME_IMPULSE_MIN)
	                AND (#statDeltaTimeImpulse <= #TIME_IMPULSE_MAX))
	                AND (#statImpulseDetected = True)
	            THEN
	                #statImpulseDetected := False;
	                #statFrameImulseDetected := true;
	            END_IF;
	            
	            //Channel detection
	            
	            IF #statFrameImulseDetected = TRUE
	            THEN
	                #statFrameImulseDetected := FALSE;
	                
	                IF #statCountChannelPos = 4
	                THEN
	                    #statCurrentPos1 := #statCountChannelPos;
	                    #statTimeImpulseSave1 := #statDeltaTimeImpulse;
	                    #statTimePauseSave1 := #statDeltaTimePause;
	                    #statTimeToImpulse := t#0ms;
	                    #statTimeToImpulse := #statTimeToImpulse + #statDeltaTimeImpulse + #statDeltaTimePause;
	                    
	                    //channel 1 ok
	                    IF (#statDeltaTimePause >= #TIME_PAUSE1_MIN)
	                        AND (#statDeltaTimePause <= #TIME_PAUSE1_MAX)
	                    THEN
	                        #statChannelActive1 := true;
	                        #statCountChannelPos := 1; // Pos 1 detected
	                    END_IF;
	                    
	                    // channel 1 not ok
	                    IF (#statDeltaTimePause >= #TIME_PAUSE2_MIN)
	                        AND (#statDeltaTimePause <= #TIME_PAUSE2_MAX)
	                    THEN
	                        #statChannelActive1 := false;
	                        #statChannelActive2 := true;
	                        #statCountChannelPos := 2; // go to next Pos 2
	                    END_IF;
	                    
	                    // channel 1 and 2 not ok
	                    IF (#statDeltaTimePause >= #TIME_PAUSE3_MIN)
	                        AND (#statDeltaTimePause <= #TIME_PAUSE3_MAX)
	                    THEN
	                        #statChannelActive1 := false;
	                        #statChannelActive2 := false;
	                        #statChannelActive3 := true;
	                        #statCountChannelPos := 2; // go to next Pos 2
	                    END_IF;
	                    
	                    // channel 1, 2 and 3 not ok
	                    IF (#statDeltaTimePause >= #TIME_PAUSE4_MIN)
	                        AND (#statDeltaTimePause <= #TIME_PAUSE4_MAX)
	                    THEN
	                        #statChannelActive1 := false;
	                        #statChannelActive2 := false;
	                        #statChannelActive3 := FALSE;
	                        #statChannelActive4 := true;
	                        #statCountChannelPos := 0;
	                    END_IF;
	                ELSIF #statCountChannelPos = 1
	                THEN
	                    #statCurrentPos2 := #statCountChannelPos;
	                    #statTimeImpulseSave2 := #statDeltaTimeImpulse;
	                    #statTimePauseSave2 := #statDeltaTimePause;
	                    #statTimeToImpulse := #statTimeToImpulse + #statDeltaTimeImpulse + #statDeltaTimePause;
	                    
	                    IF (#statDeltaTimePause >= #TIME_PAUSE1_MIN)
	                        AND (#statDeltaTimePause <= #TIME_PAUSE1_MAX)
	                    THEN
	                        #statChannelActive2 := true;
	                        #statCountChannelPos := 2; // go to next pos 2
	                    END_IF;
	                    
	                    IF (#statDeltaTimePause >= #TIME_PAUSE2_MIN)
	                        AND (#statDeltaTimePause <= #TIME_PAUSE2_MAX)
	                    THEN
	                        #statChannelActive2 := false;
	                        #statChannelActive3 := true;
	                        #statCountChannelPos := 2; // go to next Pos 2
	                    END_IF;
	                    
	                    IF (#statDeltaTimePause >= #TIME_PAUSE3_MIN)
	                        AND (#statDeltaTimePause <= #TIME_PAUSE3_MAX)
	                    THEN
	                        #statChannelActive2 := false;
	                        #statChannelActive3 := false;
	                        #statChannelActive4 := true;
	                        #statCountChannelPos := 0;
	                    END_IF;
	                ELSIF #statCountChannelPos = 2
	                THEN
	                    #statCurrentPos3 := #statCountChannelPos;
	                    #statTimeImpulseSave3 := #statDeltaTimeImpulse;
	                    #statTimePauseSave3 := #statDeltaTimePause;
	                    #statTimeToImpulse := #statTimeToImpulse + #statDeltaTimeImpulse + #statDeltaTimePause;
	                    
	                    IF (#statDeltaTimePause >= #TIME_PAUSE1_MIN)
	                        AND (#statDeltaTimePause <= #TIME_PAUSE1_MAX)
	                    THEN
	                        #statChannelActive3 := true;
	                        #statCountChannelPos := 3; // go to next pos 3
	                    END_IF;
	                    
	                    IF (#statDeltaTimePause >= #TIME_PAUSE2_MIN)
	                        AND (#statDeltaTimePause <= #TIME_PAUSE2_MAX)
	                    THEN
	                        #statChannelActive3 := false;
	                        #statChannelActive4 := true;
	                        #statCountChannelPos := 0;
	                    END_IF;
	                ELSIF #statCountChannelPos = 3
	                THEN
	                    #statCurrentPos4 := #statCountChannelPos;
	                    #statTimeImpulseSave4 := #statDeltaTimeImpulse;
	                    #statTimePauseSave4 := #statDeltaTimePause;
	                    #statTimeToImpulse := #statTimeToImpulse + #statDeltaTimeImpulse + #statDeltaTimePause;
	                    
	                    IF (#statDeltaTimePause >= #TIME_PAUSE1_MIN)
	                        AND (#statDeltaTimePause <= #TIME_PAUSE1_MAX)
	                    THEN
	                        #statChannelActive4 := true;
	                    END_IF;
	                    #statCountChannelPos := 0; // go to pos 0
	                END_IF;
	            END_IF;
	            
	        #STATE_ERROR:
	            #error := true;
	            #busy := false;
	            #done := false;
	            #statSysTimerStart := false;
	            #statWatchDogTimerStartR := false;
	            #statWatchDogTimerStartF := false;
	            #status := #statStatus;
	            #statStatus := w#16#0000;
	            #statIndex := #STATE_IDLE;
	        ELSE  // Statement section ELSE
	            #statIndex := #STATE_IDLE;
	    END_CASE;
	    
	    #instWatchDogTimerR(IN := #statWatchDogTimerStartR,
	                       PT := t#6s);
	    #statWatchDogTimerRunR:= #instWatchDogTimerR.ET;
	    
	    
	    #instWatchDogTimerF(IN := #statWatchDogTimerStartF,
	                       PT := t#6s); 
	    #statWatchDogTimerRunF:= #instWatchDogTimerF.ET;
	          
	    #instSysTimer(IN := #statSysTimerStart,
	                  PT := T#4s);
	    #statSysTimerRun:= #instSysTimer.ET; 
	    
	    IF  (#instWatchDogTimerR.Q = true)
	        OR (#instWatchDogTimerF.Q = true)
	        THEN
	        #statIndex := #STATE_ERROR;
	        #statStatus := 16#8002;
	    END_IF;
	      
	    
	    IF #instSysTimer.Q=true
	    THEN
	        #statIndex := #STATE_ERROR;
	        #statStatus := 16#8001;
	    END_IF;
	    
	    //Edge control
	    #statImpulseOld := #impulse;
	    #statResetOld := #reset;
	    
	    // Cycle time control
	    #statSysTimeOld := #statSysTime;
	
END_FUNCTION_BLOCK

FUNCTION "FC450_ALARM_DECODING_WINCC" : Void
{ S7_Optimized_Access := 'TRUE' }
VERSION : 0.1
   VAR_TEMP 
      i : Int;
      val1 : Int;
   END_VAR


BEGIN
	// IF THE SIZE OF 'DB426_ALARMS_WARNINGS' IS CHANGED, THE MAXIMUM NUMBER OF WORDS 
	// IN THE 'FOR' LOOP AND THE NUMBER OF BYTES TRANSFERRED FROM 'DB426' TO 'DB429' WITH BLKMOV MUST BE UPDATED.
	
	#val1 := BLKMOV(SRCBLK := P#DB426.DBX0.0 BYTE 3874, DSTBLK => P#DB430.DBX0.0 BYTE 3874);
	
	FOR #i := 0 TO 1937 DO
	    "DB430_ALARMS_WARNINGS_WINCC_AUX".Alarms[#i] := SWAP("DB430_ALARMS_WARNINGS_WINCC_AUX".Alarms[#i]);
	END_FOR;
	
	#val1 := BLKMOV(SRCBLK := P#DB430.DBX0.0 Byte 3874, DSTBLK => P#DB429.DBX0.0 BYTE 3874);
END_FUNCTION

FUNCTION "FC2401_DTL_TO_UNIX_TIME_1" : Word
{ S7_Optimized_Access := 'TRUE' }
VERSION : 0.1
   VAR_INPUT 
      SYSTEM_TIME_DTL {InstructionName := 'DTL'; LibVersion := '1.0'} : DTL;
   END_VAR

   VAR_OUTPUT 
      UNIX_TIME_SEC : UDInt;
      UNIX_TIME_MSEC : UDInt;
   END_VAR

   VAR_TEMP 
      UNIX_TIME_UDINT : UDInt;
      NANOSEC_REAL : Real;
      MILISEC_REAL : Real;
   END_VAR

   VAR CONSTANT 
      DELTA_1970_1990 : UDInt := 631_152_000;
      SEC_PER_DAY : UDInt := 86400;
   END_VAR


BEGIN
	#FC2401_DTL_TO_UNIX_TIME_1 := 1;
	
	// Convert the system time value to Dint
	#UNIX_TIME_UDINT := (DATE_TO_UDINT(DTL_TO_DATE(#SYSTEM_TIME_DTL)) * #SEC_PER_DAY) + (TOD_TO_UDINT(DTL_TO_TOD(#SYSTEM_TIME_DTL)) / 1000) + #DELTA_1970_1990;
	
	// System nanoseconds converted to miliseconds
	#NANOSEC_REAL := UDINT_TO_REAL(#SYSTEM_TIME_DTL.NANOSECOND);
	#MILISEC_REAL := #NANOSEC_REAL / 1000000.0;
	
	// Conversion to  Output
	#UNIX_TIME_SEC := #UNIX_TIME_UDINT;
	#UNIX_TIME_MSEC := REAL_TO_UDINT(#MILISEC_REAL);
	
	// Done convertion
	#FC2401_DTL_TO_UNIX_TIME_1 := 0;
END_FUNCTION

FUNCTION_BLOCK "FB7238_VARIABLES_PLC_HMI_GENERAL"
{ S7_Optimized_Access := 'TRUE' }
VERSION : 0.1
   VAR_INPUT DB_SPECIFIC
      FEEDERS_MANUAL_MODE : Bool;
      FEEDERS_AUTO_MODE : Bool;
      HOPPERS_MANUAL_MODE : Bool;
      HOPPERS_AUTO_MODE : Bool;
   END_VAR

   VAR_OUTPUT 
      FEEDERS_MODE_STATE : Int;
      HOPPERS_MODE_STATE : Int;
   END_VAR


BEGIN
	(*
	PLC TO HMI
	*)
	// UNIT 01 MODE STATE
	IF #FEEDERS_MANUAL_MODE = TRUE  AND #FEEDERS_AUTO_MODE = FALSE THEN
	    // Statement section IF
	    #FEEDERS_MODE_STATE := 3;
	ELSIF #FEEDERS_MANUAL_MODE = FALSE  AND #FEEDERS_AUTO_MODE = TRUE THEN
	    #FEEDERS_MODE_STATE := 1;
	END_IF;
	
	
	// UNIT 02 MODE STATE
	IF #HOPPERS_MANUAL_MODE = TRUE AND #HOPPERS_AUTO_MODE = FALSE THEN
	    // Statement section IF
	    #HOPPERS_MODE_STATE := 3;
	ELSIF #HOPPERS_MANUAL_MODE = FALSE AND #HOPPERS_AUTO_MODE = TRUE THEN
	    #HOPPERS_MODE_STATE := 1;
	END_IF;
	
	
	
	
END_FUNCTION_BLOCK

DATA_BLOCK "DB21205_UNIT_01_COMBINER_MEDICOAT"   // DB21205
{ DB_Accessible_From_OPC_UA := 'FALSE' }
VERSION : 0.1
// stored: AutoNumber false, DBAccessibleFromOPCUA false, DBAccessibleFromWebserver true, InstanceOfName FB21200_POWDER_FLOW_SENSOR_MEDICOAT, InstanceOfType FB
"FB21200_POWDER_FLOW_SENSOR_MEDICOAT"
BEGIN
END_DATA_BLOCK

DATA_BLOCK "DB21206_UNIT_02_COMBINER_MEDICOAT"   // DB21206
{ DB_Accessible_From_OPC_UA := 'FALSE' }
VERSION : 0.1
// stored: AutoNumber false, DBAccessibleFromOPCUA false, DBAccessibleFromWebserver true, InstanceOfName FB21200_POWDER_FLOW_SENSOR_MEDICOAT, InstanceOfType FB
"FB21200_POWDER_FLOW_SENSOR_MEDICOAT"
BEGIN
END_DATA_BLOCK

DATA_BLOCK "DB21209_UNIT_01_LASER_HEAD_MEDICOAT"   // DB21209
{ DB_Accessible_From_OPC_UA := 'FALSE' }
VERSION : 0.1
// stored: AutoNumber false, DBAccessibleFromOPCUA false, DBAccessibleFromWebserver true, InstanceOfName FB21200_POWDER_FLOW_SENSOR_MEDICOAT, InstanceOfType FB
"FB21200_POWDER_FLOW_SENSOR_MEDICOAT"
BEGIN
END_DATA_BLOCK

DATA_BLOCK "DB21210_UNIT_02_LASER_HEAD_MEDICOAT"   // DB21210
{ DB_Accessible_From_OPC_UA := 'FALSE' }
VERSION : 0.1
// stored: AutoNumber false, DBAccessibleFromOPCUA false, DBAccessibleFromWebserver true, InstanceOfName FB21200_POWDER_FLOW_SENSOR_MEDICOAT, InstanceOfType FB
"FB21200_POWDER_FLOW_SENSOR_MEDICOAT"
BEGIN
END_DATA_BLOCK

DATA_BLOCK "DB21222_POWDER_FILLING_START_STOP_BY_CURRENT_DB"   // DB21222
{ DB_Accessible_From_OPC_UA := 'FALSE' }
VERSION : 0.1
// stored: AutoNumber false, DBAccessibleFromOPCUA false, DBAccessibleFromWebserver true, InstanceOfName FB21222_POWDER_FILLING_START_STOP_BY_CURRENT, InstanceOfType FB
"FB21222_POWDER_FILLING_START_STOP_BY_CURRENT"
BEGIN
END_DATA_BLOCK

DATA_BLOCK "DB21225_HOPPER_1_POWDER_FILLING_START_STOP_BY_CURRENT_DB"   // DB21225
{ DB_Accessible_From_OPC_UA := 'FALSE' }
VERSION : 0.1
// stored: AutoNumber false, DBAccessibleFromOPCUA false, DBAccessibleFromWebserver true, InstanceOfName FB21222_POWDER_FILLING_START_STOP_BY_CURRENT, InstanceOfType FB
"FB21222_POWDER_FILLING_START_STOP_BY_CURRENT"
BEGIN
END_DATA_BLOCK

DATA_BLOCK "DB21226_HOPPER_2_POWDER_FILLING_START_STOP_BY_CURRENT_DB"   // DB21226
{ DB_Accessible_From_OPC_UA := 'FALSE' }
VERSION : 0.1
// stored: AutoNumber false, DBAccessibleFromOPCUA false, DBAccessibleFromWebserver true, InstanceOfName FB21222_POWDER_FILLING_START_STOP_BY_CURRENT, InstanceOfType FB
"FB21222_POWDER_FILLING_START_STOP_BY_CURRENT"
BEGIN
END_DATA_BLOCK

DATA_BLOCK "DB21991_LGF_FloatingAverage_Start"   // DB21991
{ DB_Accessible_From_OPC_UA := 'FALSE' }
AUTHOR : Siemens_Digital_Industry
FAMILY : LGF
NAME : LGF_FloatingAverage
VERSION : 0.1
// stored: AutoNumber false, DBAccessibleFromOPCUA false, DBAccessibleFromWebserver true, InstanceOfName FB21990_LGF_FloatingAverage, InstanceOfType FB
"FB21990_LGF_FloatingAverage"
   // VAR_INPUT
   //    cyclicExecution : Bool;
   //    trigger : Bool;
   //    value : LReal;
   //    windowSize : Int;
   //    reset : Bool;
   // END_VAR
   // VAR_OUTPUT
   //    average { ExternalWritable := 'False'} : LReal;
   //    windowSizeReached { ExternalWritable := 'False'} : Bool;
   //    error { ExternalWritable := 'False'} : Bool;
   //    status { ExternalWritable := 'False'} : Word;
   // END_VAR
   // VAR
   //    statValues { ExternalAccessible := 'False'; ExternalVisible := 'False'; ExternalWritable := 'False'} : Array[0..100] of LReal;
   //    statValuesSum { ExternalAccessible := 'False'; ExternalVisible := 'False'; ExternalWritable := 'False'} : LReal;
   //    statArithmeticAverage { ExternalAccessible := 'False'; ExternalVisible := 'False'; ExternalWritable := 'False'} : LReal;
   //    statWindowSizeOld { ExternalAccessible := 'False'; ExternalVisible := 'False'; ExternalWritable := 'False'} : Int;
   //    statCounter { ExternalAccessible := 'False'; ExternalVisible := 'False'; ExternalWritable := 'False'} : Int;
   //    statwindowSizeReached { ExternalAccessible := 'False'; ExternalVisible := 'False'; ExternalWritable := 'False'} : Bool;
   //    statTriggerOld { ExternalAccessible := 'False'; ExternalVisible := 'False'; ExternalWritable := 'False'} : Bool;
   // END_VAR
BEGIN
END_DATA_BLOCK

DATA_BLOCK "DB21992_LGF_FloatingAverage_Stop"   // DB21992
{ DB_Accessible_From_OPC_UA := 'FALSE' }
AUTHOR : Siemens_Digital_Industry
FAMILY : LGF
NAME : LGF_FloatingAverage
VERSION : 0.1
// stored: AutoNumber false, DBAccessibleFromOPCUA false, DBAccessibleFromWebserver true, InstanceOfName FB21990_LGF_FloatingAverage, InstanceOfType FB
"FB21990_LGF_FloatingAverage"
   // VAR_INPUT
   //    cyclicExecution : Bool;
   //    trigger : Bool;
   //    value : LReal;
   //    windowSize : Int;
   //    reset : Bool;
   // END_VAR
   // VAR_OUTPUT
   //    average { ExternalWritable := 'False'} : LReal;
   //    windowSizeReached { ExternalWritable := 'False'} : Bool;
   //    error { ExternalWritable := 'False'} : Bool;
   //    status { ExternalWritable := 'False'} : Word;
   // END_VAR
   // VAR
   //    statValues { ExternalAccessible := 'False'; ExternalVisible := 'False'; ExternalWritable := 'False'} : Array[0..100] of LReal;
   //    statValuesSum { ExternalAccessible := 'False'; ExternalVisible := 'False'; ExternalWritable := 'False'} : LReal;
   //    statArithmeticAverage { ExternalAccessible := 'False'; ExternalVisible := 'False'; ExternalWritable := 'False'} : LReal;
   //    statWindowSizeOld { ExternalAccessible := 'False'; ExternalVisible := 'False'; ExternalWritable := 'False'} : Int;
   //    statCounter { ExternalAccessible := 'False'; ExternalVisible := 'False'; ExternalWritable := 'False'} : Int;
   //    statwindowSizeReached { ExternalAccessible := 'False'; ExternalVisible := 'False'; ExternalWritable := 'False'} : Bool;
   //    statTriggerOld { ExternalAccessible := 'False'; ExternalVisible := 'False'; ExternalWritable := 'False'} : Bool;
   // END_VAR
BEGIN
END_DATA_BLOCK

DATA_BLOCK "DB2002_BA_MODES_MG1"   // DB2002
{ DB_Accessible_From_OPC_UA := 'FALSE' }
VERSION : 0.1
// stored: AutoNumber false, DBAccessibleFromOPCUA false, DBAccessibleFromWebserver true, InstanceOfName FB2002_BA_MODE, InstanceOfType FB
"FB2002_BA_MODE"
BEGIN
END_DATA_BLOCK

DATA_BLOCK "DB2003_BA_MODES_MG2"   // DB2003
{ DB_Accessible_From_OPC_UA := 'FALSE' }
VERSION : 0.1
// stored: AutoNumber false, DBAccessibleFromOPCUA false, DBAccessibleFromWebserver true, InstanceOfName FB2002_BA_MODE, InstanceOfType FB
"FB2002_BA_MODE"
BEGIN
END_DATA_BLOCK

DATA_BLOCK "DB2003_CNC_MODES_MG1"   // DB2003
{ DB_Accessible_From_OPC_UA := 'FALSE' }
VERSION : 0.1
// stored: AutoNumber false, DBAccessibleFromOPCUA false, DBAccessibleFromWebserver false, InstanceOfName FB2003_CNC_MODES, InstanceOfType FB
"FB2003_CNC_MODES"
BEGIN
END_DATA_BLOCK

DATA_BLOCK "DB2005_CNC_MODES_MG2"   // DB2005
VERSION : 0.1
// stored: AutoNumber false, DBAccessibleFromOPCUA true, DBAccessibleFromWebserver true, InstanceOfName FB2003_CNC_MODES, InstanceOfType FB
"FB2003_CNC_MODES"
BEGIN
END_DATA_BLOCK

DATA_BLOCK "DB2005_MDA_MODE_MG1"   // DB2005
{ DB_Accessible_From_OPC_UA := 'FALSE' }
VERSION : 0.1
// stored: AutoNumber false, DBAccessibleFromOPCUA false, DBAccessibleFromWebserver false, InstanceOfName FB2005_MDA_MODE, InstanceOfType FB
"FB2005_MDA_MODE"
BEGIN
END_DATA_BLOCK

DATA_BLOCK "DB2006_REFERENCE_MODE_MG1"   // DB2006
{ DB_Accessible_From_OPC_UA := 'FALSE' }
VERSION : 0.1
// stored: AutoNumber false, DBAccessibleFromOPCUA false, DBAccessibleFromWebserver false, InstanceOfName FB2006_REFERENCE_MODE, InstanceOfType FB
"FB2006_REFERENCE_MODE"
BEGIN
END_DATA_BLOCK

DATA_BLOCK "DB2007_INCREMENTAL_MODE_MG1"   // DB2007
{ DB_Accessible_From_OPC_UA := 'FALSE' }
VERSION : 0.1
// stored: AutoNumber false, DBAccessibleFromOPCUA false, DBAccessibleFromWebserver false, InstanceOfName FB2007_INCREMENTAL_MODE, InstanceOfType FB
"FB2007_INCREMENTAL_MODE"
BEGIN
END_DATA_BLOCK

DATA_BLOCK "DB2011_AUTO_SINGLE_SEMI_MANUAL_MG1_DB"   // DB2011
{ DB_Accessible_From_OPC_UA := 'FALSE' }
VERSION : 0.1
// stored: AutoNumber false, DBAccessibleFromOPCUA false, DBAccessibleFromWebserver false, InstanceOfName FB2001_AUTO_SINGLE_SEMI_MANUAL, InstanceOfType FB
"FB2001_AUTO_SINGLE_SEMI_MANUAL"
BEGIN
END_DATA_BLOCK

DATA_BLOCK "DB2015_MDA_MODE_MG2"   // DB2015
{ DB_Accessible_From_OPC_UA := 'FALSE' }
VERSION : 0.1
// stored: AutoNumber false, DBAccessibleFromOPCUA false, DBAccessibleFromWebserver false, InstanceOfName FB2005_MDA_MODE, InstanceOfType FB
"FB2005_MDA_MODE"
BEGIN
END_DATA_BLOCK

DATA_BLOCK "DB2016_REFERENCE_MODE_MG2"   // DB2016
{ DB_Accessible_From_OPC_UA := 'FALSE' }
VERSION : 0.1
// stored: AutoNumber false, DBAccessibleFromOPCUA false, DBAccessibleFromWebserver false, InstanceOfName FB2006_REFERENCE_MODE, InstanceOfType FB
"FB2006_REFERENCE_MODE"
BEGIN
END_DATA_BLOCK

DATA_BLOCK "DB2017_INCREMENTAL_MODE_MG2"   // DB2017
{ DB_Accessible_From_OPC_UA := 'FALSE' }
VERSION : 0.1
// stored: AutoNumber false, DBAccessibleFromOPCUA false, DBAccessibleFromWebserver false, InstanceOfName FB2007_INCREMENTAL_MODE, InstanceOfType FB
"FB2007_INCREMENTAL_MODE"
BEGIN
END_DATA_BLOCK

DATA_BLOCK "DB2021_AUTO_SINGLE_SEMI_MANUAL_MG2_DB"   // DB2021
{ DB_Accessible_From_OPC_UA := 'FALSE' }
VERSION : 0.1
// stored: AutoNumber false, DBAccessibleFromOPCUA false, DBAccessibleFromWebserver false, InstanceOfName FB2001_AUTO_SINGLE_SEMI_MANUAL, InstanceOfType FB
"FB2001_AUTO_SINGLE_SEMI_MANUAL"
BEGIN
END_DATA_BLOCK

DATA_BLOCK "DB2107_MACHINE_LIGHT"   // DB2107
{ DB_Accessible_From_OPC_UA := 'FALSE' }
VERSION : 0.1
// stored: AutoNumber false, DBAccessibleFromOPCUA false, DBAccessibleFromWebserver true, InstanceOfName FB2107_LIGHTS, InstanceOfType FB
"FB2107_LIGHTS"
BEGIN
END_DATA_BLOCK

DATA_BLOCK "DB2108_UNIT_1_STATION_3_LIGHT"   // DB2108
{ DB_Accessible_From_OPC_UA := 'FALSE' }
VERSION : 0.1
// stored: AutoNumber false, DBAccessibleFromOPCUA false, DBAccessibleFromWebserver true, InstanceOfName FB2107_LIGHTS, InstanceOfType FB
"FB2107_LIGHTS"
BEGIN
END_DATA_BLOCK

DATA_BLOCK "DB2109_UNIT_2_STATION_3_LIGHT"   // DB2109
{ DB_Accessible_From_OPC_UA := 'FALSE' }
VERSION : 0.1
// stored: AutoNumber false, DBAccessibleFromOPCUA false, DBAccessibleFromWebserver true, InstanceOfName FB2107_LIGHTS, InstanceOfType FB
"FB2107_LIGHTS"
BEGIN
END_DATA_BLOCK

DATA_BLOCK "DB7001_UNIT_1_MAIN_SAFETY_DOOR"   // DB7001
{ DB_Accessible_From_OPC_UA := 'FALSE' }
AUTHOR : ETXETAR
VERSION : 1.0
// stored: AutoNumber false, DBAccessibleFromOPCUA false, DBAccessibleFromWebserver true, InstanceOfName FB7001_SAFETY_DOOR, InstanceOfType FB
"FB7001_SAFETY_DOOR"
BEGIN
END_DATA_BLOCK

DATA_BLOCK "DB7002_UNIT_1_STATION_2_SAFETY_DOOR"   // DB7002
{ DB_Accessible_From_OPC_UA := 'FALSE' }
AUTHOR : ETXETAR
VERSION : 1.0
// stored: AutoNumber false, DBAccessibleFromOPCUA false, DBAccessibleFromWebserver true, InstanceOfName FB7001_SAFETY_DOOR, InstanceOfType FB
"FB7001_SAFETY_DOOR"
BEGIN
END_DATA_BLOCK

DATA_BLOCK "DB7003_UNIT_1_STATION_4_SAFETY_DOOR"   // DB7003
{ DB_Accessible_From_OPC_UA := 'FALSE' }
AUTHOR : ETXETAR
VERSION : 1.0
// stored: AutoNumber false, DBAccessibleFromOPCUA false, DBAccessibleFromWebserver true, InstanceOfName FB7001_SAFETY_DOOR, InstanceOfType FB
"FB7001_SAFETY_DOOR"
BEGIN
END_DATA_BLOCK

DATA_BLOCK "DB7011_UNIT_2_MAIN_SAFETY_DOOR"   // DB7011
{ DB_Accessible_From_OPC_UA := 'FALSE' }
AUTHOR : ETXETAR
VERSION : 1.0
// stored: AutoNumber false, DBAccessibleFromOPCUA false, DBAccessibleFromWebserver true, InstanceOfName FB7001_SAFETY_DOOR, InstanceOfType FB
"FB7001_SAFETY_DOOR"
BEGIN
END_DATA_BLOCK

DATA_BLOCK "DB7012_UNIT_2_STATION_2_SAFETY_DOOR"   // DB7012
{ DB_Accessible_From_OPC_UA := 'FALSE' }
AUTHOR : ETXETAR
VERSION : 1.0
// stored: AutoNumber false, DBAccessibleFromOPCUA false, DBAccessibleFromWebserver true, InstanceOfName FB7001_SAFETY_DOOR, InstanceOfType FB
"FB7001_SAFETY_DOOR"
BEGIN
END_DATA_BLOCK

DATA_BLOCK "DB7013_UNIT_2_STATION_4_SAFETY_DOOR"   // DB7013
{ DB_Accessible_From_OPC_UA := 'FALSE' }
AUTHOR : ETXETAR
VERSION : 1.0
// stored: AutoNumber false, DBAccessibleFromOPCUA false, DBAccessibleFromWebserver true, InstanceOfName FB7001_SAFETY_DOOR, InstanceOfType FB
"FB7001_SAFETY_DOOR"
BEGIN
END_DATA_BLOCK
